(* CODESYS project 02_Ftp_Client.ecp

Project tree, tasks and I/O mapping:
  PFC200 : 750-8212 PFC200 G2 2ETH RS, WAGO, order no. 0750-8212, version 5.16.3.46
    application Application
      libraries: ; WagoAppFTP, 1.3.1.3 (WAGO)
      task PLC_Task (cyclic, interval 50 ms, priority 15) calls PLC_PRG
      program PLC_PRG [ST]
      DUTs/
        data type typProgress
      program PrgSampleFromLib [ST]
    ProjectConfiguration
    Kbus : Kbus, WAGO, version 1.4.0.2
        unmapped channels: K-BUS diagnostics
    MODBUS
      MODBUS : MODBUS, WAGO, order no. n/a, version 1.1.1.16
    Serial
      COM1 : COM1, WAGO, version 0.0.0.19
    Common.PCI
    EtherNet/IP
      Ethernet : Ethernet, WAGO, version 35.16.0.0
          settings: IPAddress = [192, 168, 1, 212]; SubnetMask = [0, 0, 0, 0]; MACAddress = [16#00, 16#00, 16#00, 16#00, 16#00, 16#00]; NetworkInterfaceName = 'br0'; NetworkInterfaceName = "br0"
  libraries: VisuSymbols, 3.5.17.0 (System); WagoVisuIcons, 1.1.0.4 (WAGO)
  00000000-0000-0000-0000-000000000000|C:\Users\u0100068\AppData\Local\Temp\8974f0b8bdb2430394b7f3e707461259\e868b832187f4f1a859da50215710801\Project.xml
*)

// PFC200/Application/DUTs/typProgress
{attribute 'strict'}
TYPE typProgress:	// for the state machine
(
	idle := 0,
	waiting,
	error);
END_TYPE

// PFC200/Application/PLC_PRG
PROGRAM PLC_PRG
VAR
	// a state machine
	eProgress:			typProgress;
	FtpClient:			FbFtp;
	xStart, xActiveMode, xBusy, xDone, xError: BOOL;
	sActivePort:		STRING(255);
	udiNBytesToTransfer,
	udiNBytesTransfered,
	udiActionCounter:	UDINT;
	sMessage:			STRING(INT#30);
	oR_TRIG: R_TRIG;
END_VAR

oR_TRIG(CLK:=xStart);

FtpClient(	sServer		:= '192.168.1.210',
			uiPort		:= 0,
			sUser		:= 'root',
			sPassword	:= 'wago',
			xActiveMode := xActiveMode,
//			sActivePort := sActivePort,
			tKeepAlive	:= T#5S,
			tTimeout	:= T#5S,
			xBusy		=> xBusy,
			xDone		=> xDone,
			xError		=> xError,
			udiNBytesToTransfer => udiNBytesToTransfer,
			udiNBytesTransfered => udiNBytesTransfered);

IF FtpClient.xBusy = FALSE THEN
	// state machine (deutsch: Zustandsautomat)
	CASE eProgress OF
		idle:
		sMessage := 'waiting for xStart...';
		IF oR_TRIG.Q THEN
			xStart:=FALSE;
			FtpClient.FileWrite(sLocalPath	:= '/var/www/myTextFile.txt',
								sRemotePath	:= '/ftp-server/pfc8212/myTextFile.txt',
								xCreateDirs	:= TRUE);
	
			udiActionCounter := udiActionCounter + 1;
			// check, if the write process is ready
			IF xDone THEN
				eProgress := waiting;
			END_IF
		END_IF
	
		waiting:
		IF FtpClient.xDone THEN
			xStart := FALSE;
			eProgress := idle;
		ELSIF FtpClient.xError THEN
			eProgress := error;
		END_IF

		error:
		sMessage := 'an error occured!';
	END_CASE
END_IF

END_PROGRAM

// PFC200/Application/PrgSampleFromLib
PROGRAM PrgSampleFromLib
VAR
	FbFTP:					WagoAppFTP.FbFTP;
	xBusy, xDone, xError:	BOOL;
	oStatus:				WagoSysErrorBase.FbResult;
	udiNBytesToTransfer,
	udiNBytesTransfered:	UDINT;
	iState:					INT;

	//List
	sListBuffer:	STRING(255);
	//Write
	sTxBuffer:		STRING(255) := 'Hello World!';
	//Read
	sRxBuffer:		STRING(255);
END_VAR

FbFTP(	sServer		:= '192.168.1.17',
		uiPort		:= 0,
		sUser		:= 'root',
		sPassword	:= 'wago',
		xActiveMode	:= FALSE,
		sActivePort	:= '',
		tKeepAlive	:= T#5S,
		tTimeout	:= T#5S,
		xBusy		=> xBusy,
		xDone		=> xDone,
		xError		=> xError,
		oStatus		=> oStatus,
		udiNBytesToTransfer	=> udiNBytesToTransfer,
		udiNBytesTransfered	=> udiNBytesTransfered);

IF FbFTP.xDone = TRUE THEN
	iState := iState + 1; 
ELSIF FbFTP.xError = TRUE THEN
	iState := 99; 
END_IF

IF FbFTP.xBusy = FALSE THEN
	CASE iState OF
	0:	// makes a directory listing of the user's home directory.
		FbFTP.List(	sRemotePath		:= '',
					pRxBuffer		:= ADR(sListBuffer),
					udiRxBufferSize	:= SIZEOF(sListBuffer),
					sFileSpec		:= '',
					xWithDetails	:= FALSE); 
	1:	// creates the directory ‘NewDir’ and the file ‘HelloWorld.txt’. Writes the data from sTxBuffer into the new file.
		FbFTP.FileWriteFromMem(	sRemotePath	:= 'NewDir/HelloWorld.txt',
								pTxBuffer	:= ADR(sTxBuffer),
								udiTxNBytes	:= LENGTH(sTxBuffer),
								xCreateDirs	:= TRUE); 
	2: 
	// create a new directory. A Path with ‘//’ at the begin starts in the root directory FbFTP.DirCreate(sRemotePath := ‘//root/NewDir/NewDir2’); 
	3: 
	// makes a directory. FbFTP.List(sRemotePath := ‘NewDir’, pRxBuffer := ADR(sListBuffer), udiRxBufferSize := SIZEOF(sListBuffer), sFileSpec := ‘*.txt’, xWithDetails := TRUE); 
	4: 
	// rename and replace the file. FbFTP.FileRename(sOldFileName := ‘//root/NewDir/HelloWorld.txt’, sNewFileName := ‘NewDir/NewDir2/Rename.txt’); 
	5: 
	// reads the data from the file. FbFTP.FileReadToMem(sRemotePath := ‘//root/NewDir/NewDir2/Rename.txt’, pRxBuffer := ADR(sRxBuffer), udiRxBufferSize := SIZEOF(sRxBuffer)); 
	6: 
	// removes the file. FbFTP.FileRemove(sRemotePath := ‘NewDir/NewDir2/Rename.txt’); 
	7: 
	// removes a directory FbFTP.DirRemove(sRemotePath := ‘//root/NewDir/NewDir2’); 
	8: 
	// removes a directory FbFTP.DirRemove(sRemotePath := ‘NewDir/’); 
	99: 
	// some error handling
	END_CASE

END_IF

END_PROGRAM
